FUNCTION_BLOCK PAEConveyorBelt EXTENDS PAEElevator
VAR_INPUT
END_VAR
VAR_OUTPUT
END_VAR
VAR
END_VAR

END_FUNCTION_BLOCK

(* stored: Version 1.1.0.1, ProductVersion 3.1.4020.12
   POU PAEConveyorBelt: Id {2f107bde-db07-4cea-888d-183fe8c7622e}, SpecialFunc None *)
